RoboDK station: 数字孪生CR10A-V4.rdk

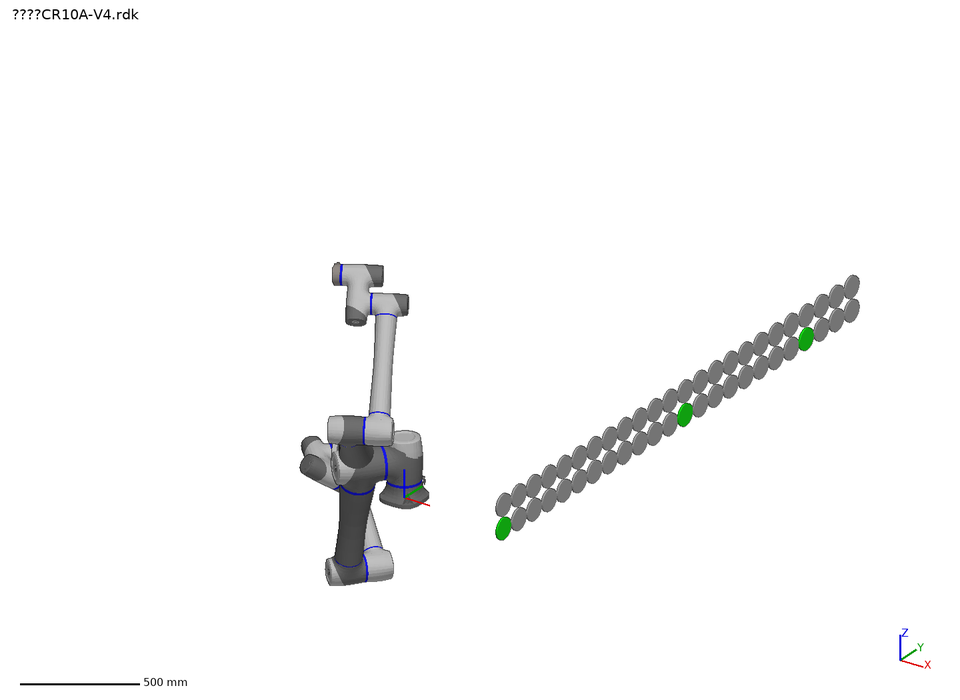
[picture v0: the station drawn from its stored meshes, robots at their saved joint values, targets as dots, program paths as lines]
Station 数字孪生V4 (saved by RoboDK 5.6.5). Poses are relative to the parent item; angles as X-Y-Z fixed-axis rotations.
  - frame DOBOT CR10 Base at (0, 0, 0) mm
    - robot DOBOT CR10: 6 axes
        modified DH rows (alpha deg, a mm, theta deg, d mm): 0, 0, 0, 176.5; 90, 0, 90, 0; 0, 607, 0, 0; 0, 568, -90, 191; -90, 0, 0, 125; 90, 0, 0, 111.4
        joint limits [-360, -360, -160, -360, -360, -360] to [360, 360, 160, 360, 360, 360]; home [0, 0, 90, 0, -90, 0]; saved at [300, 307, 100, 0, 0, 0]
  - frame DOBOT CR10(Visual) Base at (0, 0, 0) mm
    - robot DOBOT CR10(Visual): 6 axes
        modified DH rows (alpha deg, a mm, theta deg, d mm): 0, 0, 0, 176.5; 90, 0, 90, 0; 0, 607, 0, 0; 0, 568, -90, 191; -90, 0, 0, 125; 90, 0, 0, 111.4
        joint limits [-360, -360, -160, -360, -360, -360] to [360, 360, 160, 360, 360, 360]; home [0, 0, 90, 0, -90, 0]; saved at [-39.27, -198.55, -103.76, -157.09, -216, 1]
    - frame IO Base at (0, 0, 0) mm
      - object DO 1 at (500, 0, 0) mm, rotated rx 0 ry 90 rz 0 deg, size 100 x 99.5 x 10 mm, geometry from _1.stl
      - object DI 1 at (500, 0, 110) mm, rotated rx 0 ry 90 rz 0 deg, size 100 x 99.5 x 10 mm, geometry from _1.stl
      - object DO 2 at (500, 110, 0) mm, rotated rx 0 ry 90 rz 0 deg, size 100 x 99.5 x 10 mm, geometry from _1.stl
      - object DI 2 at (500, 110, 110) mm, rotated rx 0 ry 90 rz 0 deg, size 100 x 99.5 x 10 mm, geometry from _1.stl
      - object DO 3 at (500, 220, 0) mm, rotated rx 0 ry 90 rz 0 deg, size 100 x 99.5 x 10 mm, geometry from _1.stl
      - object DI 3 at (500, 220, 110) mm, rotated rx 0 ry 90 rz 0 deg, size 100 x 99.5 x 10 mm, geometry from _1.stl
      - object DO 4 at (500, 330, 0) mm, rotated rx 0 ry 90 rz 0 deg, size 100 x 99.5 x 10 mm, geometry from _1.stl
      - object DI 4 at (500, 330, 110) mm, rotated rx 0 ry 90 rz 0 deg, size 100 x 99.5 x 10 mm, geometry from _1.stl
      - object DO 5 at (500, 440, 0) mm, rotated rx 0 ry 90 rz 0 deg, size 100 x 99.5 x 10 mm, geometry from _1.stl
      - object DI 5 at (500, 440, 110) mm, rotated rx 0 ry 90 rz 0 deg, size 100 x 99.5 x 10 mm, geometry from _1.stl
      - object DO 6 at (500, 550, 0) mm, rotated rx 0 ry 90 rz 0 deg, size 100 x 99.5 x 10 mm, geometry from _1.stl
      - object DI 6 at (500, 550, 110) mm, rotated rx 0 ry 90 rz 0 deg, size 100 x 99.5 x 10 mm, geometry from _1.stl
      - object DO 7 at (500, 660, 0) mm, rotated rx 0 ry 90 rz 0 deg, size 100 x 99.5 x 10 mm, geometry from _1.stl
      - object DI 7 at (500, 660, 110) mm, rotated rx 0 ry 90 rz 0 deg, size 100 x 99.5 x 10 mm, geometry from _1.stl
      - object DO 8 at (500, 770, 0) mm, rotated rx 0 ry 90 rz 0 deg, size 100 x 99.5 x 10 mm, geometry from _1.stl
      - object DI 8 at (500, 770, 110) mm, rotated rx 0 ry 90 rz 0 deg, size 100 x 99.5 x 10 mm, geometry from _1.stl
      - object DO 9 at (500, 880, 0) mm, rotated rx 0 ry 90 rz 0 deg, size 100 x 99.5 x 10 mm, geometry from _1.stl
      - object DI 9 at (500, 880, 110) mm, rotated rx 0 ry 90 rz 0 deg, size 100 x 99.5 x 10 mm, geometry from _1.stl
      - object DO 10 at (500, 990, 0) mm, rotated rx 0 ry 90 rz 0 deg, size 100 x 99.5 x 10 mm, geometry from _1.stl
      - object DI 10 at (500, 990, 110) mm, rotated rx 0 ry 90 rz 0 deg, size 100 x 99.5 x 10 mm, geometry from _1.stl
      - object DO 11 at (500, 1100, 0) mm, rotated rx 0 ry 90 rz 0 deg, size 100 x 99.5 x 10 mm, geometry from _1.stl
      - object DI 11 at (500, 1100, 110) mm, rotated rx 0 ry 90 rz 0 deg, size 100 x 99.5 x 10 mm, geometry from _1.stl
      - object DO 12 at (500, 1210, 0) mm, rotated rx 0 ry 90 rz 0 deg, size 100 x 99.5 x 10 mm, geometry from _1.stl
      - object DI 12 at (500, 1210, 110) mm, rotated rx 0 ry 90 rz 0 deg, size 100 x 99.5 x 10 mm, geometry from _1.stl
      - object DO 13 at (500, 1320, 0) mm, rotated rx 0 ry 90 rz 0 deg, size 100 x 99.5 x 10 mm, geometry from _1.stl
      - object DI 13 at (500, 1320, 110) mm, rotated rx 0 ry 90 rz 0 deg, size 100 x 99.5 x 10 mm, geometry from _1.stl
      - object DO 14 at (500, 1430, 0) mm, rotated rx 0 ry 90 rz 0 deg, size 100 x 99.5 x 10 mm, geometry from _1.stl
      - object DI 14 at (500, 1430, 110) mm, rotated rx 0 ry 90 rz 0 deg, size 100 x 99.5 x 10 mm, geometry from _1.stl
      - object DO 15 at (500, 1540, 0) mm, rotated rx 0 ry 90 rz 0 deg, size 100 x 99.5 x 10 mm, geometry from _1.stl
      - object DI 15 at (500, 1540, 110) mm, rotated rx 0 ry 90 rz 0 deg, size 100 x 99.5 x 10 mm, geometry from _1.stl
      - object DO 16 at (500, 1650, 0) mm, rotated rx 0 ry 90 rz 0 deg, size 100 x 99.5 x 10 mm, geometry from _1.stl
      - object DI 16 at (500, 1650, 110) mm, rotated rx 0 ry 90 rz 0 deg, size 100 x 99.5 x 10 mm, geometry from _1.stl
      - object DO 17 at (500, 1760, 0) mm, rotated rx 0 ry 90 rz 0 deg, size 100 x 99.5 x 10 mm, geometry from _1.stl
      - object DI 17 at (500, 1760, 110) mm, rotated rx 0 ry 90 rz 0 deg, size 100 x 99.5 x 10 mm, geometry from _1.stl
      - object DO 18 at (500, 1870, 0) mm, rotated rx 0 ry 90 rz 0 deg, size 100 x 99.5 x 10 mm, geometry from _1.stl
      - object DI 18 at (500, 1870, 110) mm, rotated rx 0 ry 90 rz 0 deg, size 100 x 99.5 x 10 mm, geometry from _1.stl
      - object DO 19 at (500, 1980, 0) mm, rotated rx 0 ry 90 rz 0 deg, size 100 x 99.5 x 10 mm, geometry from _1.stl
      - object DI 19 at (500, 1980, 110) mm, rotated rx 0 ry 90 rz 0 deg, size 100 x 99.5 x 10 mm, geometry from _1.stl
      - object DO 20 at (500, 2090, 0) mm, rotated rx 0 ry 90 rz 0 deg, size 100 x 99.5 x 10 mm, geometry from _1.stl
      - object DI 20 at (500, 2090, 110) mm, rotated rx 0 ry 90 rz 0 deg, size 100 x 99.5 x 10 mm, geometry from _1.stl
      - object DO 21 at (500, 2200, 0) mm, rotated rx 0 ry 90 rz 0 deg, size 100 x 99.5 x 10 mm, geometry from _1.stl
      - object DI 21 at (500, 2200, 110) mm, rotated rx 0 ry 90 rz 0 deg, size 100 x 99.5 x 10 mm, geometry from _1.stl
      - object DO 22 at (500, 2310, 0) mm, rotated rx 0 ry 90 rz 0 deg, size 100 x 99.5 x 10 mm, geometry from _1.stl
      - object DI 22 at (500, 2310, 110) mm, rotated rx 0 ry 90 rz 0 deg, size 100 x 99.5 x 10 mm, geometry from _1.stl
      - object DO 23 at (500, 2420, 0) mm, rotated rx 0 ry 90 rz 0 deg, size 100 x 99.5 x 10 mm, geometry from _1.stl
      - object DI 23 at (500, 2420, 110) mm, rotated rx 0 ry 90 rz 0 deg, size 100 x 99.5 x 10 mm, geometry from _1.stl
      - object DO 24 at (500, 2530, 0) mm, rotated rx 0 ry 90 rz 0 deg, size 100 x 99.5 x 10 mm, geometry from _1.stl
      - object DI 24 at (500, 2530, 110) mm, rotated rx 0 ry 90 rz 0 deg, size 100 x 99.5 x 10 mm, geometry from _1.stl
  - Python program 数字孪生V4 (listed below)

--- Python program 数字孪生V4 ---
import tkinter as tk
from tkinter import messagebox, scrolledtext
import threading
import numpy as np
import socket
from robolink import *  # RoboDK API
from robodk import *    # Robot toolbox
from dobot_apiV4 import DobotApiDashboard, DobotApiFeedBack, MyType


class RoboDKDOBOTUI:
    def __init__(self, master):
        self.master = master
        master.title("DOBOT RoboDK UI")
        master.geometry("800x950")

        self.rdk = Robolink()
        self.robot = self.rdk.Item("DOBOT CR10")
        self.robot_visual = self.rdk.Item("DOBOT CR10(Visual)")

        self.dashboard = None
        self.feedback = None
        self.connected = False

        self.step = 0.5

        self.di_label = tk.StringVar()
        self.do_label = tk.StringVar()
        self.do_vars = [tk.IntVar(value=0) for _ in range(8)]
        self.status_label = tk.StringVar(value="未连接")

        self.joint_target = [tk.DoubleVar(value=0.0) for _ in range(6)]
        self.cartesian_target = [tk.DoubleVar(value=0.0) for _ in range(6)]

        self.joint_current = [tk.StringVar() for _ in range(6)]
        self.cartesian_current = [tk.StringVar() for _ in range(6)]

        self.log_text = None

        self.build_ui()
        self.sync_cartesian_from_visual()  # 启动时同步笛卡尔

    def build_ui(self):
        tk.Label(self.master, text="IP地址:").grid(row=0, column=0)
        self.ip_entry = tk.Entry(self.master)
        self.ip_entry.insert(0, "192.168.5.1")
        self.ip_entry.grid(row=0, column=1)

        tk.Button(self.master, text="连接", command=self.connect).grid(row=0, column=2)
        tk.Button(self.master, text="MovJ", command=self.send_movj).grid(row=0, column=3)
        tk.Button(self.master, text="MovL", command=self.send_movl).grid(row=0, column=4)
        tk.Button(self.master, text="清除报警", command=self.clear_error).grid(row=0, column=5)

        tk.Label(self.master, text="机器人状态:").grid(row=1, column=0)
        tk.Label(self.master, textvariable=self.status_label, fg="blue").grid(row=1, column=1, columnspan=3)

        row_base = 2
        tk.Label(self.master, text="当前角度:").grid(row=row_base, column=0, pady=(10,0))
        for i in range(6):
            tk.Label(self.master, text=f"J{i+1}:").grid(row=row_base+1, column=i)
            tk.Label(self.master, textvariable=self.joint_current[i]).grid(row=row_base+2, column=i)

        tk.Label(self.master, text="当前笛卡尔:").grid(row=row_base+3, column=0, pady=(10,0))
        for i, name in enumerate(["X","Y","Z","Rx","Ry","Rz"]):
            tk.Label(self.master, text=name).grid(row=row_base+4, column=i)
            tk.Label(self.master, textvariable=self.cartesian_current[i]).grid(row=row_base+5, column=i)

        tk.Label(self.master, text="期待角度:").grid(row=row_base+6, column=0, pady=(10,0))
        for i in range(6):
            tk.Label(self.master, text=f"J{i+1}:").grid(row=row_base+7, column=i)
            tk.Entry(self.master, textvariable=self.joint_target[i], width=6).grid(row=row_base+8, column=i)
            tk.Button(self.master, text="+", command=lambda i=i: self.adjust_target_joint(i, self.step)).grid(row=row_base+9, column=i)
            tk.Button(self.master, text="-", command=lambda i=i: self.adjust_target_joint(i, -self.step)).grid(row=row_base+10, column=i)

        tk.Label(self.master, text="期待笛卡尔:").grid(row=row_base+11, column=0, pady=(10,0))
        for i, name in enumerate(["X","Y","Z","Rx","Ry","Rz"]):
            tk.Label(self.master, text=name).grid(row=row_base+12, column=i)
            tk.Entry(self.master, textvariable=self.cartesian_target[i], width=6).grid(row=row_base+13, column=i)

        tk.Label(self.master, text="DI:").grid(row=row_base+14, column=0)
        tk.Label(self.master, textvariable=self.di_label).grid(row=row_base+14, column=1, columnspan=4)

        tk.Label(self.master, text="DO:").grid(row=row_base+15, column=0)
        tk.Label(self.master, textvariable=self.do_label).grid(row=row_base+15, column=1, columnspan=4)

        tk.Label(self.master, text="DO设置:").grid(row=row_base+16, column=0)
        for i in range(8):
            tk.Checkbutton(self.master, text=f"DO{i+1}", variable=self.do_vars[i], command=lambda i=i: self.set_do(i + 1, self.do_vars[i].get())).grid(row=row_base+16+i//4, column=1+i%4)

        tk.Label(self.master, text="日志:").grid(row=row_base+19, column=0)
        self.log_text = scrolledtext.ScrolledText(self.master, height=10, width=80)
        self.log_text.grid(row=row_base+20, column=0, columnspan=6, padx=5, pady=5)

    def log(self, text):
        self.log_text.insert(tk.END, text + "\n")
        self.log_text.see(tk.END)

    def connect(self):
        if self.connected:
            self.dashboard.close()
            self.feedback.close()
            self.connected = False
            self.status_label.set("未连接")
            self.log("已断开连接")
            return

        ip = self.ip_entry.get()
        try:
            self.dashboard = DobotApiDashboard(ip, 29999)
            self.feedback = DobotApiFeedBack(ip, 30004)
            self.feedback.socket_dobot.setsockopt(socket.SOL_SOCKET, socket.SO_RCVBUF, 1440)
            self.connected = True
            self.status_label.set("已连接，检查中...")
            self.log("连接成功")
            threading.Thread(target=self.update_feedback, daemon=True).start()
        except Exception as e:
            messagebox.showerror("错误", str(e))
            self.log("连接失败: " + str(e))

    def update_feedback(self):
        while self.connected:
            data = b''
            hasRead = 0
            while hasRead < 1440:
                temp = self.feedback.socket_dobot.recv(1440 - hasRead)
                if temp:
                    data += temp
                    hasRead += len(temp)
            a = np.frombuffer(data, dtype=MyType)
            if hex(a['test_value'][0]) == '0x123456789abcdef':
                q = a["q_actual"][0] if "q_actual" in a.dtype.names else [0]*6
                tool = a["tool_vector_actual"][0] if "tool_vector_actual" in a.dtype.names else [0]*6

                for i in range(6):
                    self.joint_current[i].set(f"{q[i]:.2f}")
                    self.cartesian_current[i].set(f"{tool[i]:.2f}")

                if self.robot_visual.Valid():
                    self.robot_visual.setJoints(q.tolist())
                if self.robot.Valid():
                    self.robot.setJoints(q.tolist())

                self.di_label.set(bin(a["digital_input_bits"][0])[2:].rjust(24, '0'))
                do_bits = bin(a["digital_output_bits"][0])[2:].rjust(24, '0')
                self.do_label.set(do_bits)
                self.update_rdk_do_visual(do_bits)

                error_code = a['error_status'][0] if 'error_status' in a.dtype.names else 0
                if error_code != 0:
                    self.status_label.set(f"错误状态：代码 {error_code}")
                else:
                    self.status_label.set("正常运行")

    def update_rdk_do_visual(self, do_bits):
        for i in range(min(24, len(do_bits))):
            item = self.rdk.Item(f"DO {i+1}")
            if item.Valid():
                if do_bits[i] == '1':
                    item.setColor([0.0, 1.0, 0.0, 1.0])
                else:
                    item.setColor([0.7, 0.7, 0.7, 1.0])

    def adjust_target_joint(self, idx, delta):
        self.joint_target[idx].set(round(self.joint_target[idx].get() + delta, 2))
        new_joints = [v.get() for v in self.joint_target]
        if self.robot_visual.Valid():
            self.robot_visual.setJoints(new_joints)
            pose = self.robot_visual.Pose().Pos()
            rpy = self.robot_visual.Pose().Rot3D()
            values = pose + rpy
            for i in range(6):
                self.cartesian_target[i].set(round(values[i], 2))

    def sync_cartesian_from_visual(self):
        if self.robot_visual.Valid():
            values = Pose_2_TxyzRxyz(self.robot_visual.Pose())
            for i in range(6):
                self.cartesian_target[i].set(round(values[i], 2))
            self.log("已从 Visual 模型同步笛卡尔")
        else:
            self.log("Visual 模型无效")

    def send_movj(self):
        if not self.connected:
            return
        angles = [v.get() for v in self.joint_target]
        self.dashboard.EnableRobot()
        result = self.dashboard.MovJ(*angles, 1)
        self.log("MovJ角度: " + str(angles))
        self.log("返回: " + result)

    def send_movl(self):
        if not self.connected:
            return
        pose = [v.get() for v in self.cartesian_target]
        self.dashboard.EnableRobot()
        result = self.dashboard.MovL(*pose, 1)
        self.log("MovL笛卡尔: " + str(pose))
        self.log("返回: " + result)

    def set_do(self, index, status):
        if not self.connected:
            return
        result = self.dashboard.DOInstant(index, status)
        self.log(f"设置 DO{index} 为 {status}: {result}")
        item = self.rdk.Item(f"DO {index}")
        if item.Valid():
            if status == 1:
                item.setColor([0.0, 1.0, 0.0, 1.0])
            else:
                item.setColor([0.7, 0.7, 0.7, 1.0])

    def clear_error(self):
        if not self.connected:
            return
        result = self.dashboard.ClearError()
        self.log("清除报警: " + result)


if __name__ == '__main__':
    root = tk.Tk()
    app = RoboDKDOBOTUI(root)
    root.mainloop()
